// TIA Portal project "used on a prototype" (V14)
// for a Greek client

(* hardware
DEVICE "HMI_2"  TP900 Comfort
   slot 0: "TP900 Comfort"  TP900 Comfort  6AV2 124-0JC01-0AX0  14.0.1.0
   slot 1: "HMI_RT_2"  TP900 Comfort  6AV2 124-0JC01-0AX0  14.0.1.0
   slot 5: "HMI_2.IE_CP_1"  PROFINET Interface  14.0.1.0
      slot 1: "PROFINET Interface_1"  PROFINET Interface
         slot 1: "Port_1"  Port
         slot 2: "Port_2"  Port
   slot 7: "HMI_2.MPI/DP_CP_1"  MPI/DP Interface  14.0.1.0
DEVICE "S7-1200 station_1"  S7-1200 Station
   slot 0: "Rack_0"  S7-1200 Rack  Rack  V1.0
   slot 1: "PLC_1"  CPU 1214C AC/DC/Rly  6ES7 214-1BG40-0XB0  V4.2
   slot 2: "AnalogIns 8xRTD_2"  SM 1231 AI8 x RTD  6ES7 231-5PF32-0XB0  V2.0
*)

// ===== PLC "PLC_1"  CPU 1214C AC/DC/Rly =====

VAR_GLOBAL   // PLC tag table "Tag table_1"
   "ConnOk" AT %MW8000 : Int;
END_VAR

ORGANIZATION_BLOCK "Main"   // OB1, LAD, ProgramCycle
TITLE = "Main Program Sweep (Cycle)"
{ S7_Optimized_Access := 'TRUE' }
VERSION : 0.1
   VAR_INPUT
      Initial_Call : Bool;   // Initial call of this OB
      Remanence : Bool;   // =True, if remanent data are available
   END_VAR
BEGIN
END_ORGANIZATION_BLOCK

ORGANIZATION_BLOCK "Cyclic interrupt_500"   // OB30, FBD, CyclicInterrupt
{ S7_Optimized_Access := 'TRUE' }
VERSION : 0.1
   VAR_INPUT
      Initial_Call : Bool;   // Initial call of this OB
      Event_Count : Int;   // Events discarded
   END_VAR
BEGIN

REGION Network 1
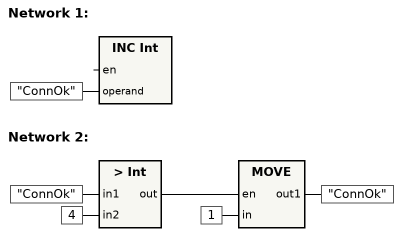
   "ConnOk" := "ConnOk" + 1;
END_REGION

REGION Network 2
   IF "ConnOk" > 4 THEN "ConnOk" := 1; END_IF;
END_REGION
END_ORGANIZATION_BLOCK

ORGANIZATION_BLOCK "Cyclic interrupt_Ds"   // OB31, SCL, CyclicInterrupt
{ S7_Optimized_Access := 'TRUE' }
VERSION : 0.1
   VAR_INPUT
      Initial_Call : Bool;   // Initial call of this OB
      Event_Count : Int;   // Events discarded
   END_VAR
BEGIN
END_ORGANIZATION_BLOCK

(* ===== HMI "HMI_RT_2" =====
system functions are stored by id; their names below are inferred from use
connection "HMI_Connection_1": ETHERNET, S7_1200_OMS

HMI tags "Default tag table"
   "Tag_ScreenNumber" : UInt, internal
   "ConnOk" : Int = PLC ConnOk AT %MW8000, 500 ms
   "ConnOk_pre" : Int, internal

screen "Root screen" 800x420, template "Template_1"
   on GenerateScreen: SetTag("Tag_ScreenNumber", 1)
   TextField "HmiScreenItemData" at 80,167 size 640x22; Text 'Welcome to HMI_2 (TP900 Comfort)!'

Template "Template_1" 800x420
   Button "Exit" at 720,360 size 78x58; TextOff 'Exit'; PictureOff "ExitRuntime_TP900_Comfort_TR"; PictureOn "ExitRuntime_TP900_Comfort_TR"
      on Release: StopRuntime(0)
   Button "Template_Button" at 640,360 size 78x58; TextOff 'Text'; PictureOff "1512075872583_1"
      on Release: ActivateScreen("Diagnostics", 0)
   Button "Template_Button_1" at 560,360 size 78x58; TextOff 'Text'; PictureOff "Right_Arrow"
   Button "Template_Button_2" at 480,360 size 78x58; TextOff 'Text'; PictureOff "Left_Arrow"
   Button "Template_Button_3" at 400,360 size 78x58; TextOff 'Text'
   Button "Template_Button_4" at 321,360 size 78x58; TextOff 'Text'
   Button "Template_Button_5" at 241,360 size 78x58; TextOff 'Text'
   Button "Template_Button_6" at 161,360 size 78x58; TextOff 'Text'
   Button "Template_Button_7" at 81,360 size 78x58; TextOff 'Text'
   Button "Start screen" at 1,360 size 78x58; TextOff 'Start screen'; PictureOff "NavigateHome_TP900_Comfort_TR"; PictureOn "NavigateHome_TP900_Comfort_TR"
      on Release: ActivateScreen("Root screen", 0)

screen "Diagnostics" 800x420
   TextField "Text field_1" at 0,5 size 800x30; Text 'AnalogIns 8xRTD_2'
   Button "Start screen" at 1,360 size 78x58; TextOn 'Start screen'; TextOff 'Start screen'; PictureOn "NavigateHome_TP900_Comfort_TR"; PictureOff "NavigateHome_TP900_Comfort_TR"
      on Release: ActivateScreen("Root screen", 0)
   IOField "I/O field_1" at 90,370 size 100x40; FormatPattern 99999
      ProcessValue <- "Tag_ScreenNumber"
   Button "Template_Button_1" at 560,360 size 78x58; TextOff 'Text'; PictureOff "Right_Arrow"
   Button "Template_Button_2" at 480,360 size 78x58; TextOff 'Text'; PictureOff "Left_Arrow"
      on Release: ActivateScreen("System diagnostics", 0)

screen "System diagnostics" 800x420
   SysDiagControl "System diagnostics view_1" at 0,0 size 800x360
   Button "Start screen" at 1,360 size 78x58; TextOn 'Start screen'; TextOff 'Start screen'; PictureOn "NavigateHome_TP900_Comfort_TR"; PictureOff "NavigateHome_TP900_Comfort_TR"
      on Release: ActivateScreen("Root screen", 0)
   Button "Template_Button_1" at 560,360 size 78x58; TextOff 'Text'; PictureOff "Right_Arrow"
      on Release: ActivateScreen("Diagnostics", 0)
   Button "Template_Button_2" at 480,360 size 78x58; TextOff 'Text'; PictureOff "Left_Arrow"

VB script "VBFunction_1"
   'Tip:
   ' 1. Use the <CTRL+SPACE> or <CTRL+I> shortcut to open a list of all objects and functions
   ' 2. Write the code using the HMI Runtime object.
   '  Example: HmiRuntime.Screens("Screen_1").
   ' 3. Use the <CTRL+J> shortcut to create an object reference.
   'Write the code as of this position:
   
   
   
   ConnOk_pre=ConnOk
*)